FUNCTION_BLOCK AxesMoveRelativeProcess EXTENDS BaseProcess
VAR_INPUT
	///Arguments to be set, before writing do_request TRUE
	{attribute 'OPC.UA.DA' := '1'}
	set: AxesMoveRelativeProcessArgs;
END_VAR
VAR_OUTPUT
	///Arguments in use by the process, if do_request was accepted
	{attribute 'OPC.UA.DA' := '1'}
	{attribute 'OPC.UA.DA.Access' := '1'}
	get: AxesMoveRelativeProcessArgs;
END_VAR
VAR_IN_OUT
END_VAR
VAR
END_VAR

IF do_request THEN
    do_request_result := request(
    units := set.units,
    value := set.value);
    do_request := FALSE;
END_IF;
SUPER^();

{attribute 'TcRpcEnable' := '1'}
METHOD start
VAR_INPUT
	///Units of the 'value' argument (RADIANS, DEGREES, ARCSECONDS, ...)
	units: AxesMoveUnits;
	///Move the axis with this value (which units depends on the 'units' argument)
	value: LREAL;
END_VAR
VAR_OUTPUT
END_VAR
VAR_IN_OUT
END_VAR
VAR
END_VAR
THIS^.get.units := units;
THIS^.get.value := value;
THIS^.statuses.busyStatus( isBusy := TRUE );
THIS^.statuses.healthStatus( isGood := TRUE );
END_METHOD

{attribute 'TcRpcEnable' := '1'}
METHOD request : RequestResults
VAR_INPUT
	///Units of the 'value' argument (RADIANS, DEGREES, ARCSECONDS, ...)
	units: AxesMoveUnits;
	///Move the axis with this value (which units depends on the 'units' argument)
	value: LREAL;
END_VAR
VAR_OUTPUT
END_VAR
VAR_IN_OUT
END_VAR
VAR
END_VAR
IF THIS^.statuses.enabledStatus.enabled THEN
    THIS^.start(
        units := units,
        value := value);
    request := RequestResults.ACCEPTED;
ELSE
    request := RequestResults.REJECTED;
END_IF;
END_METHOD

END_FUNCTION_BLOCK

(* stored: Version 1.1.0.1, ProductVersion 3.1.4019.2
   POU AxesMoveRelativeProcess: Id {ab1536d4-4e05-4045-a393-8dc116fede54}, SpecialFunc None
   Method start: Id {03fa504b-5fed-412e-b70a-e0c5d9e5c81a}
   Method request: Id {66be002b-1e20-4776-9547-c116df6b4ad6} *)
